FUNCTION_BLOCK E_CTU (* Basic FB with empty ECC *)
  (* Standard: 61499-2 *)
  (* Version 1.0, 2016-05-26, AZ, fortiss GmbH *)
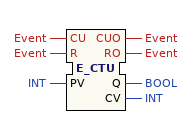
  EVENT_INPUT
    CU;
    R;
  END_EVENT
  EVENT_OUTPUT
    CUO;
    RO;
  END_EVENT
  VAR_INPUT
    PV : INT;
  END_VAR
  VAR_OUTPUT
    Q : BOOL;
    CV : INT;
  END_VAR
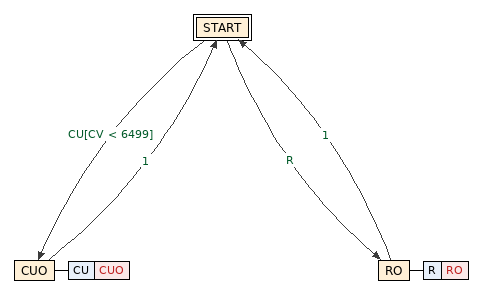
  EC_STATES
    START;
    RO : R -> RO;
    CUO : CU -> CUO;
  END_STATES
  EC_TRANSITIONS
    START TO CUO := CU[CV < 6499];
    START TO RO := R;
    RO TO START := 1;
    CUO TO START := 1;
  END_TRANSITIONS
  ALGORITHM R IN ST:
CV := 0;&#13;&#10;Q := FALSE;
  END_ALGORITHM
  ALGORITHM CU IN ST:
CV := CV + 1;&#13;&#10;Q  := (CV &gt;= PV);
  END_ALGORITHM
END_FUNCTION_BLOCK
